INTERFACE I_Mc2Axis_PTP EXTENDS I_Mc2Axis, I_Axis_PTP

END_INTERFACE

(* stored: Version 1.1.0.1, ProductVersion 3.1.4026.20
   Itf I_Mc2Axis_PTP: Id {bfe1ba3a-5906-4db0-8de5-4bed3b573cf8} *)
